Fanuc KAREL source: kt00899.KL

-- PROVISIONAL review KL for V1013-1; original PC SHA256 c6696dc4c7db538e7af64d69450a81d8ad6da117d131268b93a41de99b440742
-- Incomplete behavior may be omitted. Consult companion uncertainty JSON. Do not deploy.
PROGRAM KT00899
%NOLOCKGROUP
VAR
  OUT : BOOLEAN
-- UNRESOLVED_DECL P1 type=000102
-- UNRESOLVED_DECL P2 type=000102
BEGIN
  -- UNRESOLVED_PC offsets 5-20; opcodes 2E,22,32,35
  -- UNRESOLVED_PC offsets 25-40; opcodes 2E,22,32,35
  -- UNRESOLVED_PC offsets 45-60; opcodes 2E,22,32,35
  -- UNRESOLVED_PC offsets 65-80; opcodes 2E,22,32,35
  -- UNRESOLVED_PC offsets 85-111; opcodes 27,27,49,7E,AD,27,9D,76,23
  -- UNRESOLVED_PC offsets 116-120; opcodes 7F
END KT00899
